{attribute addProperty BoxType "EL3611-1030-0016"}
{attribute addProperty Id "AI_InputsAT %I*AI_Inputs_BED3E98C4860WcStateAT %I*WcState_98A4DF7520.250InfoDataAT %I*InfoData_BC63D37F80100"}
{attribute addProperty CRC "1773532003"}
{attribute addProperty SizeInBites "130"}
{attribute addProperty SizeInBytes "16.25"}
TYPE EL3611_AB57A9CF :
STRUCT
	{attribute addProperty Name "AI_Inputs"}
	AI_Inputs : AI_Inputs_BED3E98C;
	{attribute addProperty Name "WcState"}
	WcState : WcState_98A4DF75;
	{attribute addProperty Name "InfoData"}
	InfoData : InfoData_BC63D37F;
END_STRUCT
END_TYPE

(* stored: Version 1.2.0.0, ProductVersion 3.1.4024.9
   DUT EL3611_AB57A9CF: Id {9330b8e0-c849-40eb-af2a-25754eea68da} *)
